FUNCTION_BLOCK ToVoltageConverter
VAR_INPUT
	in	:	LREAL;
	
	negative	:	LREAL;
END_VAR
VAR_OUTPUT
	voltage	:	INT;
END_VAR
VAR
END_VAR

IF in > 0 THEN
	voltage := LREAL_TO_INT(in/10 * 32767);
ELSIF in < 0 THEN
	voltage := LREAL_TO_INT(in/10 * 32768);
ELSIF in = 0 THEN
	voltage := 0;
END_IF

END_FUNCTION_BLOCK

(* stored: Version 1.1.0.1, ProductVersion 3.1.4024.12
   POU ToVoltageConverter: Id {e6a8335b-afa3-4761-ade4-7a458d67fc80}, SpecialFunc None *)
